// TIA Portal V18 export
DATA_BLOCK "Valuestobelogged"   // DB57
{ S7_Optimized_Access := 'TRUE' }
VERSION : 0.1
// stored: AutoNumber true, DBAccessibleFromOPCUA true, IsOnlyStoredInLoadMemory false, IsRetainMemResEnabled false, IsWriteProtectedInAS false, MemoryReserve 100
   VAR
      Datatobelogged : Struct
         Variable01_Bool : Bool;
         Variable02_Bool : Bool;
         Variable03_Dint : DInt;
         Variable04_Dint : DInt;
         Variable05_Dint : DInt;
         Variable06_Dint : DInt;
      END_STRUCT;
      LogColumns : String := 'Column01, Column02, Column03, Column04, Column05, Column06';
   END_VAR
BEGIN
END_DATA_BLOCK
